PROGRAM Motion
VAR
	FB_Power: MC_Power;
	FB_Stop: MC_Stop;
	FB_StopPuller: MC_Stop;
	FB_StopPullerVirtual: MC_Stop;
	FB_Velocity: MC_MoveVelocity;
	FB_VelocityPuller: MC_MoveVelocity;
	FB_Relative: MC_MoveRelative;
	FB_ReadStatus: MC_ReadStatus;
	FB_Reset: MC_Reset;
	FB_Manual: MC_Jog;
	FB_Power2: MC_Power;
	FB_Power3: MC_Power;
	FB_GearInVelo: MC_GearInVelo;
	FB_GearOut: MC_GearOut;
	FB_ManualPuller: MC_Jog;
END_VAR

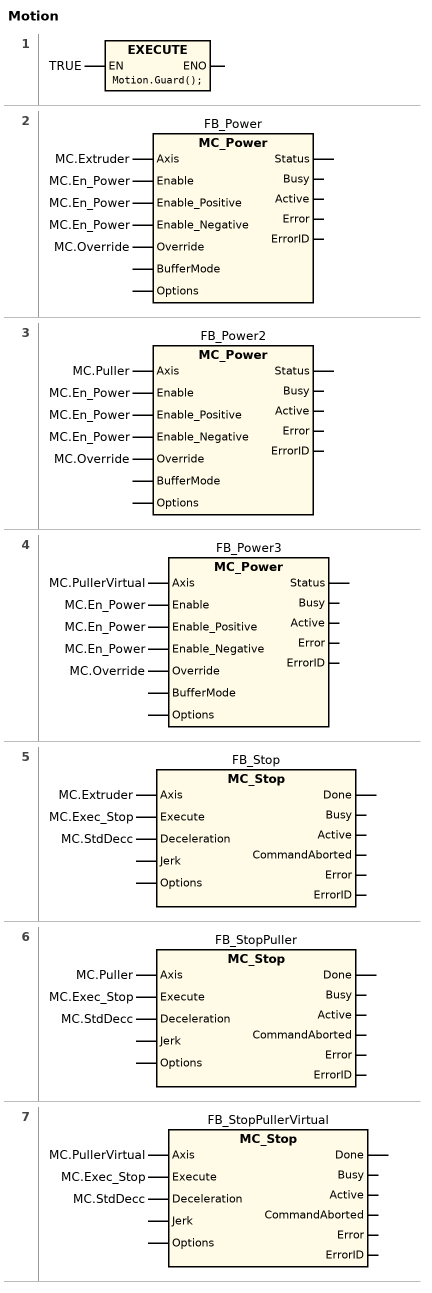
// NETWORK 1
Motion.Guard();

// NETWORK 2
FB_Power(
    Axis := MC.Extruder,
    Enable := MC.En_Power,
    Enable_Positive := MC.En_Power,
    Enable_Negative := MC.En_Power,
    Override := MC.Override); // MC_Power

// NETWORK 3
FB_Power2(
    Axis := MC.Puller,
    Enable := MC.En_Power,
    Enable_Positive := MC.En_Power,
    Enable_Negative := MC.En_Power,
    Override := MC.Override); // MC_Power

// NETWORK 4
FB_Power3(
    Axis := MC.PullerVirtual,
    Enable := MC.En_Power,
    Enable_Positive := MC.En_Power,
    Enable_Negative := MC.En_Power,
    Override := MC.Override); // MC_Power

// NETWORK 5
FB_Stop(Axis := MC.Extruder, Execute := MC.Exec_Stop, Deceleration := MC.StdDecc); // MC_Stop

// NETWORK 6
FB_StopPuller(Axis := MC.Puller, Execute := MC.Exec_Stop, Deceleration := MC.StdDecc); // MC_Stop

// NETWORK 7
FB_StopPullerVirtual(Axis := MC.PullerVirtual, Execute := MC.Exec_Stop, Deceleration := MC.StdDecc); // MC_Stop

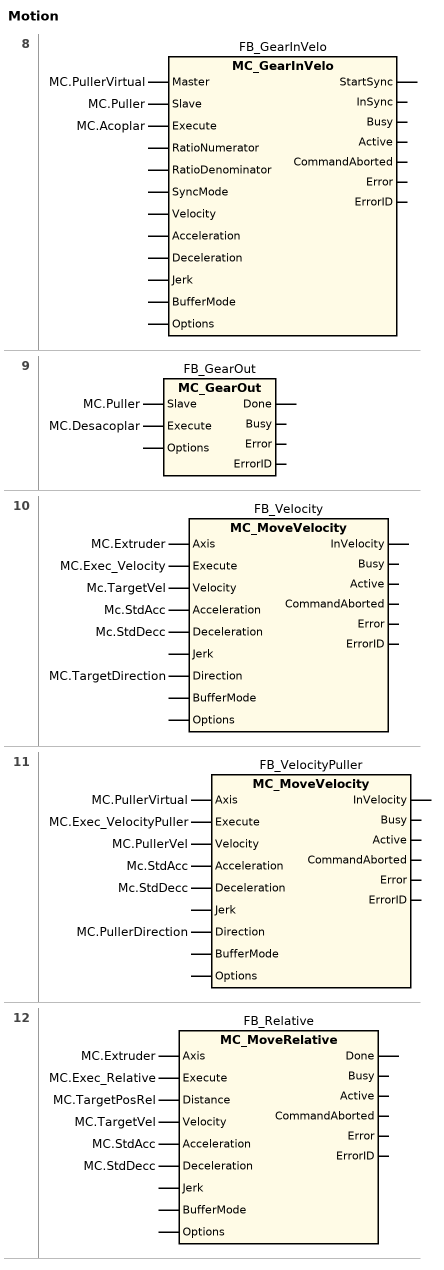
// NETWORK 8
FB_GearInVelo(Master := MC.PullerVirtual, Slave := MC.Puller, Execute := MC.Acoplar); // MC_GearInVelo

// NETWORK 9
FB_GearOut(Slave := MC.Puller, Execute := MC.Desacoplar); // MC_GearOut

// NETWORK 10
FB_Velocity(
    Axis := MC.Extruder,
    Execute := MC.Exec_Velocity,
    Velocity := Mc.TargetVel,
    Acceleration := Mc.StdAcc,
    Deceleration := Mc.StdDecc,
    Direction := MC.TargetDirection); // MC_MoveVelocity

// NETWORK 11
FB_VelocityPuller(
    Axis := MC.PullerVirtual,
    Execute := MC.Exec_VelocityPuller,
    Velocity := MC.PullerVel,
    Acceleration := Mc.StdAcc,
    Deceleration := Mc.StdDecc,
    Direction := MC.PullerDirection); // MC_MoveVelocity

// NETWORK 12
FB_Relative(
    Axis := MC.Extruder,
    Execute := MC.Exec_Relative,
    Distance := MC.TargetPosRel,
    Velocity := MC.TargetVel,
    Acceleration := MC.StdAcc,
    Deceleration := MC.StdDecc); // MC_MoveRelative

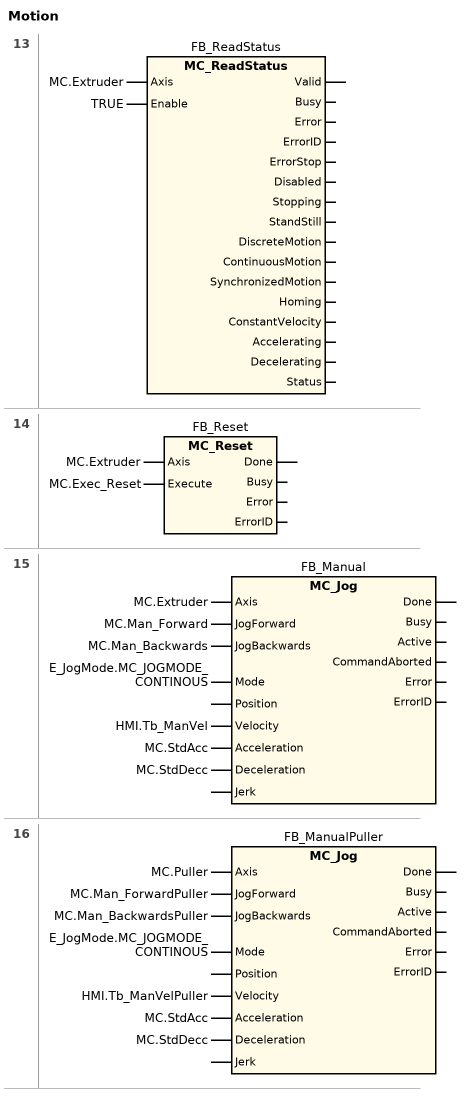
// NETWORK 13
FB_ReadStatus(Axis := MC.Extruder, Enable := TRUE); // MC_ReadStatus

// NETWORK 14
FB_Reset(Axis := MC.Extruder, Execute := MC.Exec_Reset); // MC_Reset

// NETWORK 15
FB_Manual(
    Axis := MC.Extruder,
    JogForward := MC.Man_Forward,
    JogBackwards := MC.Man_Backwards,
    Mode := E_JogMode.MC_JOGMODE_CONTINOUS,
    Velocity := HMI.Tb_ManVel,
    Acceleration := MC.StdAcc,
    Deceleration := MC.StdDecc); // MC_Jog

// NETWORK 16
FB_ManualPuller(
    Axis := MC.Puller,
    JogForward := MC.Man_ForwardPuller,
    JogBackwards := MC.Man_BackwardsPuller,
    Mode := E_JogMode.MC_JOGMODE_CONTINOUS,
    Velocity := HMI.Tb_ManVelPuller,
    Acceleration := MC.StdAcc,
    Deceleration := MC.StdDecc); // MC_Jog

ACTION Guard:
MC.Exec_Reset:=FALSE;
IF HMI.Bt_ResetAxis THEN
	IF MC.Extruder.Status.Error = TRUE THEN
		MC.Exec_Reset:= TRUE;
	END_IF
END_IF
END_ACTION

ACTION InitMotion:
MC.En_Power := FALSE;
MC.Exec_Relative := FALSE;
MC.Exec_Stop := FALSE;
MC.Exec_Velocity := FALSE;
MC.Exec_VelocityPuller:=FALSE;
MC.Acoplar:=FALSE;
MC.Desacoplar:=FALSE;
IO.Q_VisionLight := FALSE;
END_ACTION

END_PROGRAM

(* stored: Version 1.1.0.1, ProductVersion 3.1.4024.9
   POU Motion: Id {d206c616-e0b3-44bf-898b-092307161bef}, SpecialFunc None
   Action Guard: Id {f5c6939b-5a7a-4a2a-b555-85eeb0c19c75}
   Action InitMotion: Id {9d46ed5d-55f9-4643-b0b6-d4b7f5e5ed0d} *)
